PROGRAM MAIN
VAR
	safe_err_ack AT %Q* : BOOL;
	safe_run AT %Q* : BOOL;
	safe_reset AT %Q* : BOOL;
	
	com_check_pub AT %Q* : BOOL;
	com_check_sub AT %I* : BOOL;
	
END_VAR

END_PROGRAM

(* stored: Version 1.1.0.1
   POU MAIN: Id {7714da33-2d4a-4cb7-869a-08ca3cc18d03}, SpecialFunc None *)
